// Interface for binary search tree
INTERFACE I_Binary_Search_Tree EXTENDS I_Collection

// Gets the type of the data on the binary search tree
PROPERTY _Type : T_Type
GET
END_GET
END_PROPERTY

// Balances Binary Search Tree. Tree will normal auto balance every time its count is a multiple of 4
METHOD Balance
END_METHOD

(* Checks if data is contained in binary search tree *)
METHOD Find : I_Binary_Search_Tree
VAR_INPUT
	Data 	: ANY; 	// Data to remove
END_VAR
VAR_OUTPUT
	bFound 	: BOOL; 		// Indicates whether data was found. Found = TRUE, Not Found = FALSE
END_VAR
END_METHOD

(* Insert data into binary search tree *)
METHOD Insert 	: I_Binary_Search_Tree
VAR_INPUT
	Data 		: ANY; // Data to insert
END_VAR
VAR_OUTPUT
	bSuccess 	: BOOL; // Indicates whether operation was successful. Success = TRUE, Failure = FALSE
END_VAR
END_METHOD

(* Removes data from binary search tree *)
METHOD Remove : I_Binary_Search_Tree
VAR_INPUT
	Data 		: ANY; // Data to remove
END_VAR
VAR_OUTPUT
	bSuccess 	: BOOL; // Indicates whether operation was successful. Success = TRUE, Failure = FALSE
END_VAR
END_METHOD

(* Traveses the binary search tree and appends into a collection *)
METHOD Traverse : I_Binary_Search_Tree
VAR_INPUT
	eMethod 		: T_BST_Traversal; // Method to traverse the binary search tree
	ipGeneric_List 	: I_Generic_List; 		// Collection to append data to.
END_VAR
END_METHOD

END_INTERFACE

(* stored: Version 1.1.0.1, ProductVersion 3.1.4024.4
   Itf I_Binary_Search_Tree: Id {55419179-6de7-49d3-9781-3e5b195ef4ef}
   Property _Type: Id {e4613852-eb90-4f05-9b06-6f3960a5073e}
   Get Get: Id {429c017c-e856-4124-839b-8c9df367c9f9}
   Method Balance: Id {06ce1c8d-c76a-4e7b-9214-7933a467613e}
   Method Find: Id {e3ba17ef-224e-426f-bcb1-84fb9f3babe6}
   Method Insert: Id {bd596eb4-af9d-4349-942d-8a75060707ca}
   Method Remove: Id {1498a712-2459-4f01-83ff-601e7c3486db}
   Method Traverse: Id {ec82924d-83fc-47b2-ac0b-da35970eceb1} *)
